TEXTLIST StationNames
  1 = 'Station 1'
  2 = 'Station 2'
  3 = 'Station 3'
  4 = 'Station 4'
  5 = 'Station 5'
  6 = 'Station 6'
   = ''
END_TEXTLIST

(* stored: Version 1.1.0.1, ProductVersion 3.1.4024.12
   TextList StationNames: Id {23f5a359-a6a4-4101-98fe-dd45085a9d71} *)
